TYPE ST_Status :
STRUCT
	bBusy, bDone, bError	: BOOL;
	nErrorId			: UDINT;
END_STRUCT
END_TYPE

(* stored: Version 1.1.0.1, ProductVersion 3.1.4024.12
   DUT ST_Status: Id {1ec0486a-7b90-4266-b70b-32b1eb3712a4} *)
